FUNCTION CurrentF_VelocityCoeff : LREAL
VAR_INPUT
    Velocity    : LREAL;
END_VAR

CurrentF_VelocityCoeff  := EXPT((Velocity/1000),2);

END_FUNCTION

(* stored: Version 1.1.0.1
   POU CurrentF_VelocityCoeff: Id {1b258ca5-4c38-0abc-3788-dd7e914aa2ca}, SpecialFunc None *)
